// TwinCAT 3 PLC project pruebaFiltrado
// ProgramVersion: 3.1.4024.0
// libraries:
//   Tc2_Standard, * (Beckhoff Automation GmbH)
//   Tc2_System, * (Beckhoff Automation GmbH)
//   Tc3_Module, * (Beckhoff Automation GmbH)
//   VisuSymbols,3.5.10.0,System
// project tree:
//   / GlobalTextList.TcGTLO, PlcTask.TcTTO (not stored), Visualization Manager.TcVMO (not stored)
//   GVLs/ GVLvars.TcGVL
//   POUs/ MAIN.TcPOU
//   VISUs/ coloresSensorVision.TcTLO, HMI.TcVIS
// real-time tasks:
//   TASK PlcTask: cycle T#10ms, priority 20, ADS port 350

// ---- GVLs/GVLvars.TcGVL
{attribute 'qualified_only'}
VAR_GLOBAL
	
	// Cuadro
	{attribute 'OPC.UA.DA' := '1'}
	botonStart : BOOL; // boton de start
	{attribute 'OPC.UA.DA' := '1'}
	botonStop : BOOL; // boton de stop 
	{attribute 'OPC.UA.DA' := '1'}
	botonReset : BOOL; // boton de reset
	{attribute 'OPC.UA.DA' := '1'}
	setaEmergencia : BOOL; // seta de emergencia 
	{attribute 'OPC.UA.DA' := '1'}
	luzVerde : BOOL; // luz verde stack
	{attribute 'OPC.UA.DA' := '1'}
	luzAmarilla : BOOL; // luz amarilla stack
	{attribute 'OPC.UA.DA' := '1'}
	luzRoja : BOOL; // luz roja stack
	{attribute 'OPC.UA.DA' := '1'}
	luzBotonStop : BOOL; // luz integrada en boton de stop
	{attribute 'OPC.UA.DA' := '1'}
	luzBotonStart : BOOL; // luz integrada en boton de start
	{attribute 'OPC.UA.DA' := '1'}
	luzBotonReset : BOOL; // luz integrada en boton de reset
	{attribute 'OPC.UA.DA' := '1'}
	modoManual : BOOL; // Estado 0 del selector
	{attribute 'OPC.UA.DA' := '1'}
	modoAuto : BOOL; // Estado 1  del selector
	
	
	
	// Cintas
	{attribute 'OPC.UA.DA' := '1'}
	cintaVision : BOOL;
	{attribute 'OPC.UA.DA' := '1'}
	cintaRemoveVision : BOOL;
	{attribute 'OPC.UA.DA' := '1'}
	cintaBasculaPositive : BOOL;
	{attribute 'OPC.UA.DA' := '1'}
	cintaBasculaNegative : BOOL;
	{attribute 'OPC.UA.DA' := '1'}
	cintaPostBascula : BOOL;
	{attribute 'OPC.UA.DA' := '1'}
	cintaRemoveBascula : BOOL;
	{attribute 'OPC.UA.DA' := '1'}
	cintaBascula : bool;

	
	
	// Sensores
	{attribute 'OPC.UA.DA' := '1'}
	pesoBascula : REAL;
	{attribute 'OPC.UA.DA' := '1'}
 	sDifusoRemoveVision : BOOL;
	{attribute 'OPC.UA.DA' := '1'}
	sDifusoRemovePeso : BOOL;
	{attribute 'OPC.UA.DA' := '1'}
	sDifusoVision : BOOL;
 	{attribute 'OPC.UA.DA' := '1'}
	sDifusoBascula : BOOL;
	{attribute 'OPC.UA.DA' := '1'}
	sDifusoPostBascula : BOOL;
	{attribute 'OPC.UA.DA' := '1'}
 	sCilindroVision : BOOL;
	{attribute 'OPC.UA.DA' := '1'}
 	sCilindroBascula : BOOL;
	{attribute 'OPC.UA.DA' := '1'}
	sVision : DINT;
	{attribute 'OPC.UA.DA' := '1'}
	sRemoveFinal : BOOL;
	{attribute 'OPC.UA.DA' := '1'}
	sSalidaCintaVision : BOOL;
	
	
	
	// Cilindros
	{attribute 'OPC.UA.DA' := '1'}
	sCilindroVisionDelantero : BOOL;
	{attribute 'OPC.UA.DA' := '1'}
	sCilindroVisionPosterior : BOOL;
	{attribute 'OPC.UA.DA' := '1'}
	sCilindroBasculaDelantero : BOOL;
	{attribute 'OPC.UA.DA' := '1'}
	sCilindroBasculaPosterior : BOOL;
	{attribute 'OPC.UA.DA' := '1'}
 	cilindroVision : BOOL;
	{attribute 'OPC.UA.DA' := '1'}
 	cilindroBascula : BOOL;
	
	
END_VAR

// ---- POUs/MAIN.TcPOU
PROGRAM MAIN
VAR
	enclaveStart: BOOL;
	cintaRemoveVision: BOOL;
	cintaBascula: BOOL;
	cintaPostBascula: BOOL;
	cintaRemoveBascula: BOOL;
	cintaVision: BOOL;
	timerVision: TON;
	cintaBasculaPositivo:bool;
	
	descarteXcolor: BOOL;
	cilindroVision: BOOL;
	cintaDescarteVision: BOOL;
	timerBascula: TON;
	descarteXpeso: BOOL;
	cilindroBascula: BOOL;
	cintaDescarteBascula: BOOL;
	startTimerVision: BOOL;
	cintaBasculaNegativo: BOOL;
	difusoVisionAnt: bool;
	descartando: BOOL;
	flancAnteriorCilindroVision : F_TRIG;
	flancoCintaDescarte : F_TRIG;
	descratandoXpeso: BOOL;
	startTimerBascula: BOOL;
	flancoCintaDescarteBascula: F_TRIG;
	flancAnteriorCilindroBascula: F_TRIG;
	luzStart: BOOL;
	luzVerde: BOOL;
	luzAmarilla: BOOL;
	luzRoja: BOOL;
	luzStop: BOOL;
	luzReset: BOOL;
	emergencia: BOOL;
	objetoPosicionDescarteV: BOOL;
	objetoPosicionDescarteP: BOOL;
	peso: REAL;
	sinComparar: BOOL := false;
	azul: BOOL;
	metal: BOOL;
	verde: BOOL;
END_VAR

(*

1 - Si se pulsa strart -> enclave y arranque de cintas
  -	** Si se pulsa stop -> parar toda la secuencia
  
2 - Si se detecta en el sensor fotoelectrico de vision
	* Se para esa cinta 2 segundos
	* Se cogen las caracteristicas del objeto
		- Base azul : 3
		- Base verde : 6
		- Base metal : 9
	* En caso de descarte 
		- Se para cinta con el sensor delanterio del cilindro
		- Se acciona el cilindro
		- Se activa la cinta de descarte con el sensor fotoelectrico 
		  ( el tiempo de activo se sabe por vel y distancia x.ej)
 
3 - Si se detecta objeto en la cinta de pesaje (sensor fotoelectrico)
	* Se para la cinta 2 segundos
	* Se cogen als caracteristicas del objeto
		- Bases verde / azul : 7 kg
		- Base metalica : 9 kg
	* En caso de descarte
		--- Repetir proceso anterior

4 - Actualizar salidas

*)

// ------------------- PASO 1  Botones Cuadro -------------------

luzStart := FALSE;
luzStop := FALSE;
luzReset := FALSE; 

IF GVLvars.botonStart AND NOT emergencia THEN
	enclaveStart := TRUE;
	cintaVision := TRUE;
	//cintaRemoveVision := TRUE;
	cintaBascula := TRUE;
	cintaPostBascula := TRUE;
	//cintaRemoveBascula 	:= TRUE;
	luzStart := TRUE; 
	luzVerde := TRUE;
	luzAmarilla := FALSE;
	luzRoja := FALSE;
END_IF

IF NOT GVLvars.botonStop AND NOT emergencia THEN
	enclaveStart := FALSE;
	cintaVision := FALSE;
	cintaRemoveVision := FALSE;
	cintaBascula := FALSE;
	cintaPostBascula := FALSE;
	cintaRemoveBascula 	:= FALSE;
	cilindroVision := FALSE;
	cilindroBascula := FALSE;
	luzStop := TRUE; 
	luzVerde := FALSE;
	luzAmarilla := TRUE;
	luzRoja := FALSE;
END_IF



IF NOT GVLvars.setaEmergencia THEN
	enclaveStart := FALSE;
	cintaVision := FALSE;
	cintaRemoveVision := FALSE;
	cintaBascula := FALSE;
	cintaPostBascula := FALSE;
	cintaRemoveBascula 	:= FALSE;
	cilindroVision := FALSE;
	cilindroBascula := FALSE;
	luzStop := FALSE; 
	luzVerde := FALSE;
	luzAmarilla := FALSE;
	luzRoja := TRUE;
	emergencia := TRUE;
	//luzReset := TRUE;
END_IF


IF GVLvars.setaEmergencia AND emergencia THEN
	IF GVLvars.botonReset THEN
		enclaveStart := TRUE;
		luzStop := FALSE; 
		luzVerde := TRUE;
		luzAmarilla := FALSE;
		luzRoja := FALSE;
		emergencia := FALSE;
		luzReset := TRUE;
		cintaVision := TRUE;
		cintaRemoveVision := TRUE;
		cintaBascula := TRUE;
		cintaPostBascula := TRUE;
		cintaRemoveBascula 	:= TRUE;
	END_IF
END_IF


// ------------------- PASO 2 - Filtro Vision -------------------
IF enclaveStart AND NOT emergencia THEN
	
	// Detectar flanco ascendente solo una vez por detección
	IF GVLvars.sDifusoVision AND NOT difusoVisionAnt THEN
		startTimerVision := TRUE;  // Arranca el temporizador solo una vez por evento
		cintaVision := FALSE; // Se para la cinta
	END_IF
	difusoVisionAnt := GVLvars.sDifusoVision;
		
	//IF GVLvars.sDifusoVision THEN
	//cintaVision := FALSE; // Se para la cinta
	//startTimerVision := TRUE;
	timerVision(IN:=startTimerVision, PT:=T#2S);
	IF timerVision.Q THEN
		startTimerVision:=FALSE;
		// Si es color azul o metalica continua 
		IF GVLvars.sVision = 3 OR GVLvars.sVision = 9 THEN
			descarteXcolor := FALSE;
		// Se descarta la base
		ELSE
			descarteXcolor := TRUE;
		END_IF
		azul := GVLvars.sVision = 3;
		metal := GVLvars.sVision = 9;
		verde := GVLvars.sVision = 6;
		cintaVision := TRUE; // Reanuda la marcha
		
	END_IF
	
	// Si hay que descratar y se detecta objeto delante del cilindro
	IF descarteXcolor AND GVLvars.sCilindroVision THEN
		descartando := TRUE;
		
	END_IF
	
	flancAnteriorCilindroVision(CLK := GVLvars.sCilindroVision);
	flancoCintaDescarte(CLK := GVLvars.sDifusoRemoveVision);
	
	// Si tenemos que descartar y el objeto para el sensor (se situa el objeto en frente del cilindro)
	IF descartando = TRUE  AND  flancAnteriorCilindroVision.Q  THEN
		objetoPosicionDescarteV:=TRUE;
		
	END_IF
	
	
	IF objetoPosicionDescarteV THEN	
		cintaVision := FALSE;
		cilindroVision := TRUE;
		cintaRemoveVision := TRUE;	
	END_IF

	// si e objeto ya esta en la cinta de descarte se reanuda con la de vision
	IF flancoCintaDescarte.Q  THEN 
		cintaVision := TRUE;
		cilindroVision := FALSE;	
		descartando := FALSE;
		cintaRemoveVision := FALSE;
		objetoPosicionDescarteV := FALSE;
		
	END_IF

	
	
// ------------------ PASO 3 - Filtro peso -------------------

	cintaBascula := TRUE;
	
	IF GVLvars.sDifusoBascula THEN
		startTimerBascula := TRUE;  // Igual que el timer de vision: arranca el temporizador solo una vez
		cintaBascula := FALSE; // Se para la cinta
	END_IF
	
	timerBascula(IN:=startTimerBascula, PT:=T#2S);
	
	IF timerBascula.Q AND sinComparar = FALSE THEN
		startTimerBascula := FALSE;
		peso := GVLvars.pesoBascula;
		// Si el peso es mayor de un umbral se descarta
		cintaBascula := TRUE; // Reanuda la marcha
		sinComparar := TRUE;
	END_IF
	
	IF  peso > 4 THEN
		descarteXpeso := TRUE;
		sinComparar := FALSE;
	ELSE
		descarteXpeso := FALSE;
		sinComparar := FALSE;
	END_IF
		
	// Si hay que descartar y se detecta objeto delante del cilindro
	IF descarteXpeso AND GVLvars.sCilindroBascula THEN
		descratandoXpeso := TRUE;
	END_IF
	
	flancAnteriorCilindroBascula(CLK := GVLvars.sCilindroBascula);
	flancoCintaDescarteBascula(CLK := GVLvars.sDifusoRemovePeso);
	
	// Si tenemos que descartar y el objeto para el sensor
	IF descratandoXpeso = TRUE AND flancAnteriorCilindroBascula.Q THEN
		objetoPosicionDescarteP:=TRUE;
	END_IF

	IF objetoPosicionDescarteP THEN
		cintaPostBascula := FALSE;
		cilindroBascula := TRUE;
		cintaRemoveBascula := TRUE;
		
	END_IF



	
	// si el objeto ya está en la cinta de descarte, se reanuda la cinta bascula
	//IF GVLvars.sCilindroBasculaDelantero THEN
	IF flancoCintaDescarteBascula.Q THEN
		cintaPostBascula := TRUE;
		cilindroBascula := FALSE;
		descratandoXpeso := FALSE;
		descarteXpeso := FALSE;
		cintaRemoveBascula := FALSE;
		objetoPosicionDescarteP := FALSE;
	END_IF



END_IF


// ----------------- PASO 4 ------------------

// Cintas
GVLvars.cintaBascula := cintaBascula;
GVLvars.cintaPostBascula := cintaPostBascula;
GVLvars.cintaRemoveBascula := cintaRemoveBascula;
GVLvars.cintaRemoveVision := cintaRemoveVision;
GVLvars.cintaVision := cintaVision;

// Cilindros
GVLvars.cilindroBascula := cilindroBascula;
GVLvars.cilindroVision := cilindroVision;

// Cuadro
GVLvars.luzAmarilla := luzAmarilla;
GVLvars.luzRoja := luzRoja;
GVLvars.luzVerde := luzVerde;
GVLvars.luzBotonStop := luzStop;
GVLvars.luzBotonStart := luzStart;

END_PROGRAM

// ---- GlobalTextList.TcGTLO
TEXTLIST GlobalTextList
  499 = '%0.1f'
  408 = '%0.2f'
  193 = '%1.2f'
  871 = '%f'
  459 = '%g'
  989 = '%i'
  813 = '%s'
  246 = '%x.yf'
  301 = 'Color Objeto'
  270 = 'Descarte'
  942 = 'Filtrado por peso'
  104 = 'Filtrado por visión'
  801 = 'Peso'
  389 = 'Reset'
  857 = 'Seta'
  747 = 'Start'
  828 = 'Stop'
  432 = 'x.yf'
END_TEXTLIST

// ---- VISUs/coloresSensorVision.TcTLO
TEXTLIST coloresSensorVision
  3 = 'Azul'
  6 = 'Verde'
  9 = 'Metal'
  0 = '-'
   = ''
END_TEXTLIST

// ---- VISUs/HMI.TcVIS
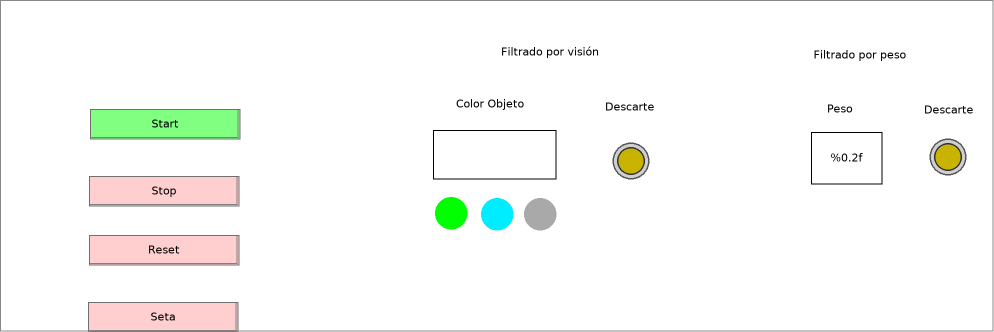
VISUALIZATION HMI  // 994x332
    Button (90,109 150x30), "Start"
        toggle GVLvars.botonStart
    Button (89,176 150x30), "Stop"
        toggle GVLvars.botonStop
    Button (89,235 150x30), "Reset"
        toggle GVLvars.botonReset
    Button (88,302 150x30), "Seta"
        toggle GVLvars.setaEmergencia
    Label (471,25 158x54), "Filtrado por visión"
    Lamp1 (610,137 42x48), variable: MAIN.descarteXcolor, style: Lamp-Lamp1-Yellow
    Label (585,92 90x30), "Descarte"
    Label (445,89 90x30), "Color Objeto"
    Label (781,28 158x54), "Filtrado por peso"
    Label (787,87 106x44), "Peso"
    Lamp1 (927,133 42x48), variable: MAIN.descratandoXpeso, style: Lamp-Lamp1-Yellow
    Label (904,95 90x30), "Descarte"
    Rectangle (433,130 123x49), text list: 'coloresSensorVision', text index: GVLvars.sVision
    Ellipse (435,197 32x32), invisible if: not Main.verde
    Ellipse (481,198 32x32), invisible if: not MAIN.azul
    Ellipse (524,198 32x32), colour toggle: MAIN.metal, invisible if: not MAIN.metal
    Rectangle (811,132 71x52), "%0.2f", text variable: MAIN.peso
END_VISUALIZATION
